// Mitsubishi GX Works2 project: motor a pasos   PLC: FX1N/FX1NC

PROGRAM MAIN
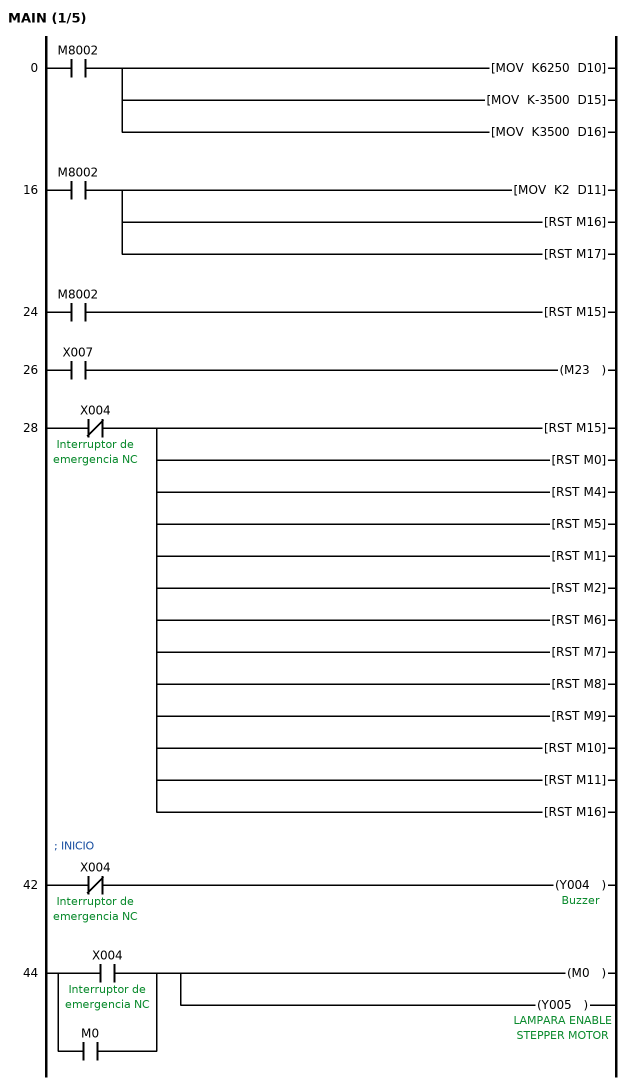
0     LD      M8002
      MOV     K6250 D10
      MOV     K-3500 D15
      MOV     K3500 D16
16    LD      M8002
      MOV     K2 D11
      RST     M16
      RST     M17
24    LD      M8002
      RST     M15
26    LD      X007
      OUT     M23
28    LDI     X004  ; Interruptor de emergencia NC
      RST     M15
      RST     M0
      RST     M4
      RST     M5
      RST     M1
      RST     M2
      RST     M6
      RST     M7
      RST     M8
      RST     M9
      RST     M10
      RST     M11
      RST     M16
; INICIO
42    LDI     X004  ; Interruptor de emergencia NC
      OUT     Y004  ; Buzzer
44    LD      X004  ; Interruptor de emergencia NC
      OR      M0
      OUT     M0
      OUT     Y005  ; LAMPARA ENABLE STEPPER MOTOR
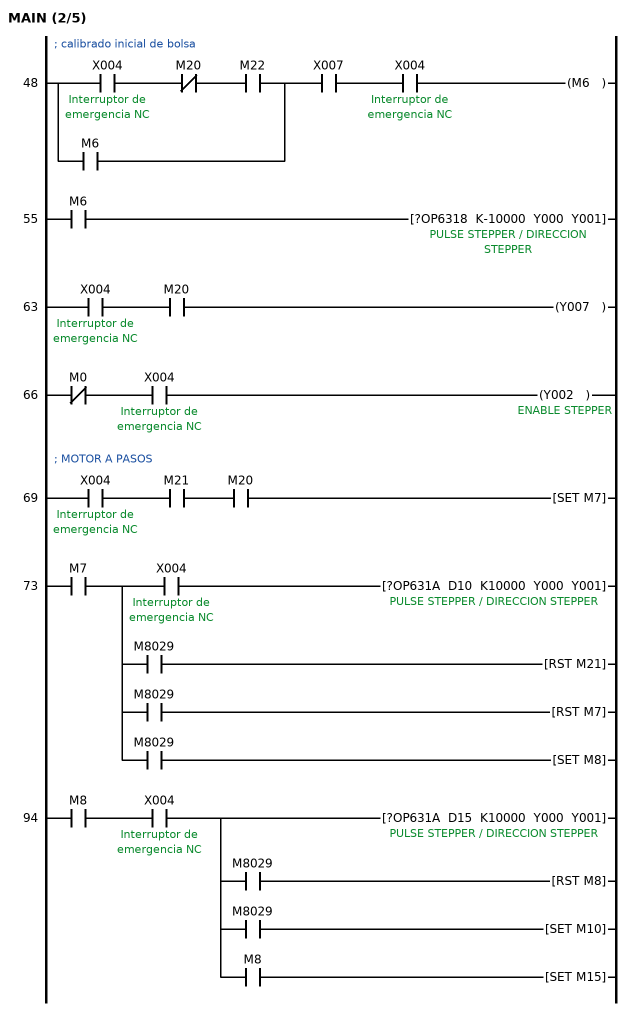
; calibrado inicial de bolsa
48    LD      X004  ; Interruptor de emergencia NC
      ANI     M20
      AND     M22
      OR      M6
      AND     X007
      AND     X004  ; Interruptor de emergencia NC
      OUT     M6
55    LD      M6
      ?OP6318 K-10000 Y000 Y001  ; PULSE STEPPER / DIRECCION STEPPER
63    LD      X004  ; Interruptor de emergencia NC
      AND     M20
      OUT     Y007
66    LDI     M0
      AND     X004  ; Interruptor de emergencia NC
      OUT     Y002  ; ENABLE STEPPER
; MOTOR A PASOS
69    LD      X004  ; Interruptor de emergencia NC
      AND     M21
      AND     M20
      SET     M7
73    LD      M7
      MPS
      AND     X004  ; Interruptor de emergencia NC
      ?OP631A D10 K10000 Y000 Y001
      MRD
      AND     M8029
      RST     M21
      MRD
      AND     M8029
      RST     M7
      MPP
      AND     M8029
      SET     M8
94    LD      M8
      AND     X004  ; Interruptor de emergencia NC
      ?OP631A D15 K10000 Y000 Y001
      MPS
      AND     M8029
      RST     M8
      MRD
      AND     M8029
      SET     M10
      MPP
      AND     M8
      SET     M15
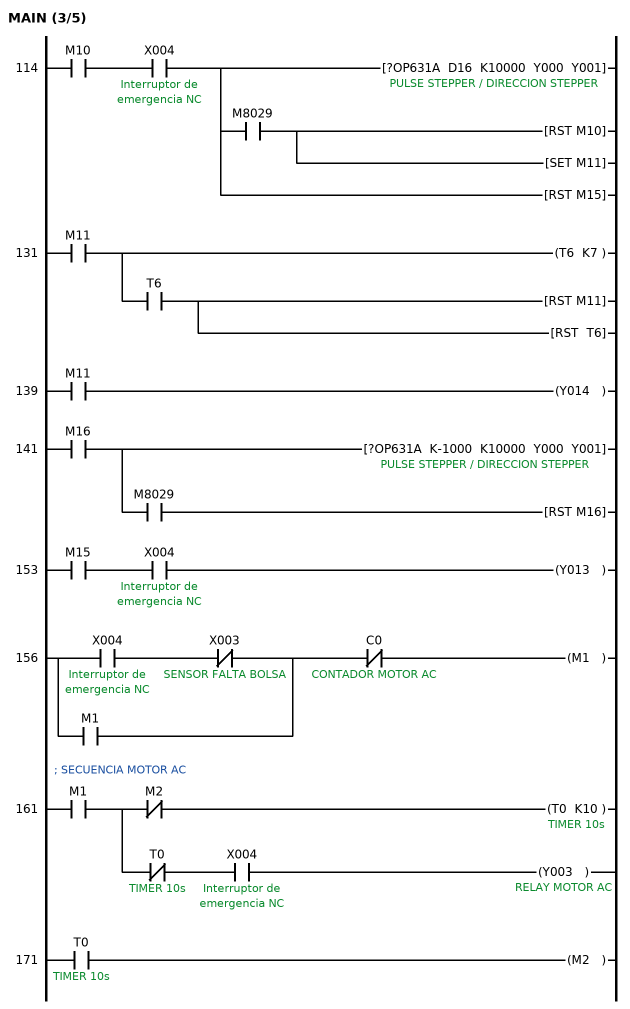
114   LD      M10
      AND     X004  ; Interruptor de emergencia NC
      ?OP631A D16 K10000 Y000 Y001
      MPS
      AND     M8029
      RST     M10
      SET     M11
      MPP
      RST     M15
131   LD      M11
      OUT     T6 K7
      AND     T6
      RST     M11
      RST     T6
139   LD      M11
      OUT     Y014
141   LD      M16
      ?OP631A K-1000 K10000 Y000 Y001
      AND     M8029
      RST     M16
153   LD      M15
      AND     X004  ; Interruptor de emergencia NC
      OUT     Y013
156   LD      X004  ; Interruptor de emergencia NC
      ANI     X003  ; SENSOR FALTA BOLSA
      OR      M1
      ANI     C0  ; CONTADOR MOTOR AC
      OUT     M1
; SECUENCIA MOTOR AC
161   LD      M1
      MPS
      ANI     M2
      OUT     T0 K10  ; TIMER 10s
      MPP
      ANI     T0  ; TIMER 10s
      AND     X004  ; Interruptor de emergencia NC
      OUT     Y003  ; RELAY MOTOR AC
171   LD      T0  ; TIMER 10s
      OUT     M2
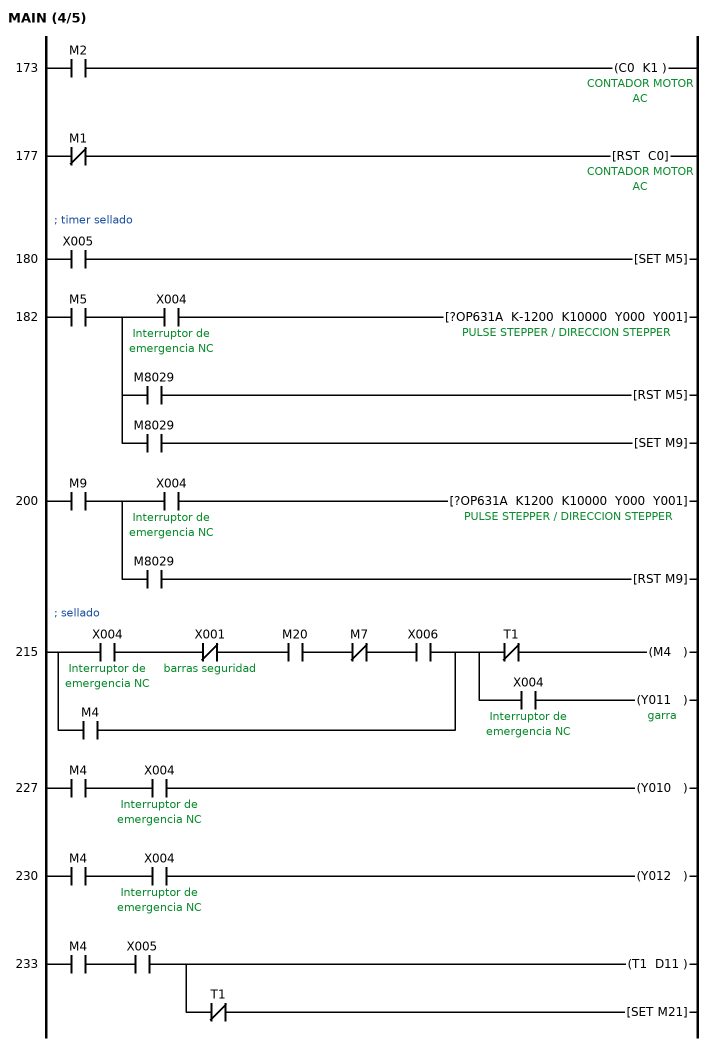
173   LD      M2
      OUT     C0 K1  ; CONTADOR MOTOR AC
177   LDI     M1
      RST     C0  ; CONTADOR MOTOR AC
; timer sellado
180   LD      X005
      SET     M5
182   LD      M5
      MPS
      AND     X004  ; Interruptor de emergencia NC
      ?OP631A K-1200 K10000 Y000 Y001
      MRD
      AND     M8029
      RST     M5
      MPP
      AND     M8029
      SET     M9
200   LD      M9
      MPS
      AND     X004  ; Interruptor de emergencia NC
      ?OP631A K1200 K10000 Y000 Y001
      MPP
      AND     M8029
      RST     M9
; sellado
215   LD      X004  ; Interruptor de emergencia NC
      ANI     X001  ; barras seguridad
      AND     M20
      ANI     M7
      AND     X006
      OR      M4
      MPS
      ANI     T1
      OUT     M4
      MPP
      AND     X004  ; Interruptor de emergencia NC
      OUT     Y011  ; garra
227   LD      M4
      AND     X004  ; Interruptor de emergencia NC
      OUT     Y010
230   LD      M4
      AND     X004  ; Interruptor de emergencia NC
      OUT     Y012
233   LD      M4
      AND     X005
      OUT     T1 D11
      ANI     T1
      SET     M21
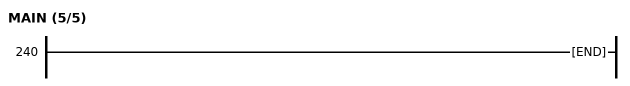
240   END
END_PROGRAM

// device comments not shown above
X002  ; DESACTIVAR MOTOR A PASOS
D0  ; REGISTRO
